Universal Robots PolyScope program: step2c_admittance_search30_z30_nostop_guard20_search2ms_line1ms_alpha70_v5.urp

Program step2c_admittance_search30_z30_nostop_guard20_search2ms_line1ms_alpha70_v5 (installation=default directory=/programs/andyl/kunwei/step2/step2c createdIn=5.11.9.1010452 lastSavedIn=5.11.9.1010452 robotSerialNumber=20225200364)
Calibrated DH parameters: a=[0.00002, -0.569483, -0.54992, -0.00001, -0.000036, 0]; d=[0.180894, -146.691669, 192.918669, -46.053088, 0.119778, 0.115602]; alpha=[1.571425, -0.001534, 0.003359, 1.568739, -1.571477, 0]; deltaTheta=[0, 0.376258, -0.101074, -0.275185, -0.000002, 0]
Robot Program (runOnlyOnce=true)
  Script file /programs/andyl/kunwei/step2/step2c/step2c/step2c_admittance_search30_z30_nostop_guard20_search2ms_line1ms_alpha70_v5.script
    | # Step2C admittance search30 v5: v4-style pre-contact approach with a 30-200 mm Z window, 50 percent lower normal admittance gain, and dynamic search-depth limit; TP-openable package.
    | # VERSION: 2026-06-08T1435HKT_STEP2C_V5_V4Z30_200_DAMP50_DEPTHFIX_NOFAILRETRACT
    | # GENERATED_AT_LOCAL: 2026-06-08T14:35:56+0800
    | # BEHAVIOR: wait for Kunwei bridge; align to old reference orientation; move to
    | # old contact-start XY; then bound the Z prep into old contact Z + 30..200 mm.
    | # If the current Z is already inside that window, keep it; otherwise move to the
    | # nearest bound and stop before search. Then search downward at 30 mm/s until 10 mm above known contact,
    | # 5 mm/s near the surface, using 2 ms speedl holds in both search and
    | # soft acquisition. Small-force early contact is gated to the near
    | # zone; far-zone unexpected contact requires larger raw force before entering
    | # soft acquisition targeting 2 N. The
    | # first 0.10 s of line control uses 10 ms speedl holds, then line control
    | # switches to 1 ms holds. Normal admittance P/I gains are reduced by 50 percent
    | # relative to the prior v4/v5 controller. Search-depth timeout is computed
    | # from the actual search-start Z so a 30-200 mm prep window can still search to
    | # 10 mm below known contact Z. A search-depth failure stops in place; it does
    | # not auto-retract upward.
    | # Aggressive normal Z correction targets signed Fz ~= -target_force_abs, where the bridge
    | # normally writes target_force_abs=5 N into input register 29.
    | # Raw contact triggers and safety guards remain unfiltered; only controller
    | # normal-velocity input uses a light force filter. No UR zero_ftsensor, no
    | # Kunwei tare/config write, no TCP/payload write, and no output register 34.
    | # Frequency contract: Kunwei raw may be about 1 kHz; RTDE handoff is requested
    | # at 500 Hz; search/admittance motion gate uses 2 ms speedl holds; line control
    | # switches to 1 ms holds after 0.10 s, but both phases must be measured before
    | # calling them 500 Hz authority. On successful completion only, retract 10 mm
    | # upward and then return to the TP-start home pose; failure paths do not auto-home.
    | 
    | def codex_abs(x):
    |   if x < 0.0:
    |     return -x
    |   end
    |   return x
    | end
    | 
    | def codex_clamp(x, lo, hi):
    |   if x < lo:
    |     return lo
    |   elif x > hi:
    |     return hi
    |   end
    |   return x
    | end
    | 
    | def codex_wait_for_sensor_ok(timeout_s):
    |   local dt = 0.002
    |   local t = 0.0
    |   while t < timeout_s:
    |     if read_input_float_register(27) > 0.5:
    |       return True
    |     end
    |     sync()
    |     t = t + dt
    |   end
    |   return False
    | end
    | 
    | def codex_wait_for_fresh_heartbeat(timeout_s):
    |   local dt = 0.002
    |   local t = 0.0
    |   local initial_heartbeat = read_input_float_register(26)
    |   local current_heartbeat = initial_heartbeat
    |   while t < timeout_s:
    |     current_heartbeat = read_input_float_register(26)
    |     write_output_float_register(26, current_heartbeat)
    |     write_output_float_register(35, 20.5)
    |     if read_input_float_register(27) > 0.5 and current_heartbeat != initial_heartbeat:
    |       return True
    |     end
    |     sync()
    |     t = t + dt
    |   end
    |   return False
    | end
    | 
    | def codex_step2_guard_stop_reason():
    |   local normal_force = read_input_float_register(24)
    |   local force_norm = read_input_float_register(25)
    |   local sensor_ok = read_input_float_register(27)
    |   local stop_request = read_input_float_register(28)
    |   local torque_norm = read_input_float_register(30)
    |   if sensor_ok < 0.5:
    |     return 3.0
    |   elif stop_request > 0.5:
    |     return 4.0
    |   elif codex_abs(normal_force) > 20.0:
    |     return 5.0
    |   elif force_norm > 50.0:
    |     return 6.0
    |   elif torque_norm > 0.6:
    |     return 7.0
    |   end
    |   return 0.0
    | end
    | 
    | def codex_write_echo(stop_reason, progress_m, correction_m, commanded_z_m_s):
    |   write_output_float_register(24, read_input_float_register(24))
    |   write_output_float_register(25, read_input_float_register(25))
    |   write_output_float_register(26, read_input_float_register(26))
    |   write_output_float_register(27, read_input_float_register(27))
    |   write_output_float_register(28, read_input_float_register(28))
    |   write_output_float_register(29, read_input_float_register(29))
    |   write_output_float_register(30, stop_reason)
    |   write_output_float_register(31, progress_m)
    |   write_output_float_register(32, correction_m)
    |   write_output_float_register(33, commanded_z_m_s)
    | end
    | 
    | def codex_step2c_full():
    |   local ux = 0.679764156
    |   local uy = -0.733430768
    |   local entry_x = 0.446585764
    |   local entry_y = 0.226717001
    |   local old_contact_z = 0.020279919
    |   local entry_z = old_contact_z + 0.100
    |   local ref_rx = 3.141572714
    |   local ref_ry = -0.000026465
    |   local ref_rz = -0.000024158
    |   local approach_speed_m_s = 0.080
    |   local approach_z_speed_m_s = 0.080
    |   local search_speed_m_s = -0.005
    |   local search_accel_m_s2 = 0.500
    |   local search_hold_s = 0.002
    |   local trigger_normal_force_n = -2.0
    |   local max_search_down_m = 0.110
    |   local stale_limit_s = 0.100
    |   local search_runtime_limit_s = 65.0
    |   local tangent_speed_m_s = 0.010
    |   local path_length_m = 0.06358
    |   local line_accel_m_s2 = 0.500
    |   local line_hold_s = 0.010
    |   local line_hold_fast_s = 0.001
    |   local line_fast_after_s = 0.100
    |   local line_runtime_limit_s = 15.0
    |   local target_force_abs_default_n = 5.0
    |   local normal_velocity_p_gain = 0.0003
    |   local normal_velocity_i_gain = 0.00004
    |   local normal_velocity_limit_m_s = 0.005
    |   local normal_filter_alpha = 0.70
    |   local integral_error_limit_n_s = 10.0
    |   local short_retract_z_m = 0.010
    |   local short_retract_speed_m_s = 0.020
    |   local home_return_speed_m_s = 0.080
    |   local stop_reason = 0.0
    |   local contact_triggered = 0
    |   local max_observed_stale_s = 0.0
    | 
    |   local home_pose = get_actual_tcp_pose()
    | 
    |   textmsg("codex step2c version 2026-06-08T1435HKT_STEP2C_V5_V4Z30_200_DAMP50_DEPTHFIX_NOFAILRETRACT start admittance_search30_v5_v4z30_200_damp50_depthfix_short_retract_home_return")
    |   write_output_float_register(35, 20.0)
    |   codex_write_echo(0.0, 0.0, 0.0, 0.0)
    | 
    |   if not codex_wait_for_fresh_heartbeat(30.0):
    |     stop_reason = 3.0
    |   end
    | 
    |   if stop_reason == 0.0:
    |     write_output_float_register(35, 21.0)
    |     local p0 = get_actual_tcp_pose()
    |     local reference_orientation_pose = p[p0[0], p0[1], p0[2], ref_rx, ref_ry, ref_rz]
    |     movel(reference_orientation_pose, a=0.030, v=approach_speed_m_s, r=0.0)
    |     stopl(0.5)
    |     write_output_float_register(35, 22.0)
    |     local p1 = get_actual_tcp_pose()
    |     local entry_xy_pose = p[entry_x, entry_y, p1[2], ref_rx, ref_ry, ref_rz]
    |     movel(entry_xy_pose, a=0.030, v=approach_speed_m_s, r=0.0)
    |     stopl(0.5)
    |     write_output_float_register(35, 23.0)
    |     local p2 = get_actual_tcp_pose()
    |     local max_entry_z = old_contact_z + 0.200
    |     local min_entry_z = old_contact_z + 0.030
    |     local bounded_entry_z = p2[2]
    |     if bounded_entry_z > max_entry_z:
    |       bounded_entry_z = max_entry_z
    |     elif bounded_entry_z < min_entry_z:
    |       bounded_entry_z = min_entry_z
    |     end
    |     if codex_abs(bounded_entry_z - p2[2]) > 0.002:
    |       local entry_pose = p[entry_x, entry_y, bounded_entry_z, ref_rx, ref_ry, ref_rz]
    |       movel(entry_pose, a=0.030, v=approach_z_speed_m_s, r=0.0)
    |       stopl(0.5)
    |     end
    |     sleep(0.20)
    |     stop_reason = codex_step2_guard_stop_reason()
    |   end
    | 
    |   if stop_reason == 0.0:
    |     write_output_float_register(35, 24.0)
    |     local search_start = get_actual_tcp_pose()
    |     max_search_down_m = search_start[2] - old_contact_z + 0.010
    |     if max_search_down_m < 0.040:
    |       max_search_down_m = 0.040
    |     elif max_search_down_m > 0.210:
    |       max_search_down_m = 0.210
    |     end
    |     local last_heartbeat = read_input_float_register(26)
    |     local stale_s = 0.0
    |     local t = 0.0
    |     local search_far_speed_m_s = -0.030
    |     local search_near_speed_m_s = -0.005
    |     local search_near_zone_m = 0.010
    |     local early_normal_force_n = -0.5
    |     local early_force_norm_n = 1.0
    |     local soft_target_force_n = 2.0
    |     local far_unexpected_normal_force_n = -5.0
    |     local far_unexpected_force_norm_n = 5.0
    |     local soft_acquire_p_gain = 0.0030
    |     local soft_velocity_limit_m_s = 0.008
    |     local soft_filter_alpha = 0.70
    |     local soft_enter_line_filtered_n = -1.8
    |     local soft_enter_line_raw_n = -2.0
    |     local soft_confirm_s = 0.030
    |     local early_contact = 0
    |     local stable_soft_s = 0.0
    |     local filtered_search_force = read_input_float_register(24)
    |     local commanded_search_z = search_far_speed_m_s
    |     while stop_reason == 0.0:
    |       local heartbeat = read_input_float_register(26)
    |       local normal_force = read_input_float_register(24)
    |       local force_norm = read_input_float_register(25)
    |       local pose_now = get_actual_tcp_pose()
    |       local search_depth_m = search_start[2] - pose_now[2]
    |       local height_above_known_contact_m = pose_now[2] - old_contact_z
    | 
    |       if heartbeat == last_heartbeat:
    |         stale_s = stale_s + search_hold_s
    |         if stale_s > max_observed_stale_s:
    |           max_observed_stale_s = stale_s
    |         end
    |       else:
    |         stale_s = 0.0
    |         last_heartbeat = heartbeat
    |       end
    | 
    |       if early_contact == 0:
    |         write_output_float_register(35, 24.0)
    |         if height_above_known_contact_m <= search_near_zone_m:
    |           if normal_force <= early_normal_force_n or force_norm > early_force_norm_n:
    |             early_contact = 1
    |             stable_soft_s = 0.0
    |             filtered_search_force = normal_force
    |             write_output_float_register(35, 24.4)
    |           end
    |         elif normal_force <= far_unexpected_normal_force_n or force_norm > far_unexpected_force_norm_n:
    |           early_contact = 1
    |           stable_soft_s = 0.0
    |           filtered_search_force = normal_force
    |           write_output_float_register(35, 24.4)
    |         end
    |       else:
    |         write_output_float_register(35, 24.4)
    |       end
    | 
    |       if stale_s > stale_limit_s:
    |         stop_reason = 2.0
    |       else:
    |         stop_reason = codex_step2_guard_stop_reason()
    |       end
    | 
    |       if stop_reason == 0.0:
    |         if search_depth_m >= max_search_down_m:
    |           stop_reason = 8.0
    |         elif t >= search_runtime_limit_s:
    |           stop_reason = 10.0
    |         else:
    |           if early_contact == 0:
    |             if height_above_known_contact_m > search_near_zone_m:
    |               commanded_search_z = search_far_speed_m_s
    |             else:
    |               commanded_search_z = search_near_speed_m_s
    |             end
    |             codex_write_echo(stop_reason, max_observed_stale_s, search_depth_m, commanded_search_z)
    |             speedl([0.0, 0.0, commanded_search_z, 0.0, 0.0, 0.0], search_accel_m_s2, search_hold_s)
    |             t = t + search_hold_s
    |           else:
    |             filtered_search_force = soft_filter_alpha * normal_force + (1.0 - soft_filter_alpha) * filtered_search_force
    |             local soft_force_error = soft_target_force_n + filtered_search_force
    |             commanded_search_z = 0.0 - codex_clamp(soft_acquire_p_gain * soft_force_error, -soft_velocity_limit_m_s, soft_velocity_limit_m_s)
    |             if filtered_search_force <= soft_enter_line_filtered_n or normal_force <= soft_enter_line_raw_n:
    |               stable_soft_s = stable_soft_s + search_hold_s
    |             else:
    |               stable_soft_s = 0.0
    |             end
    |             codex_write_echo(stop_reason, stable_soft_s, search_depth_m, commanded_search_z)
    |             if stable_soft_s >= soft_confirm_s:
    |               contact_triggered = 1
    |               stop_reason = 11.0
    |             else:
    |               speedl([0.0, 0.0, commanded_search_z, 0.0, 0.0, 0.0], search_accel_m_s2, search_hold_s)
    |               t = t + search_hold_s
    |             end
    |           end
    |         end
    |       end
    |     end
    |     stopl(0.5)
    | 
    |   end
    | 
    |   if contact_triggered == 1:
    |     stop_reason = 0.0
    |   end
    | 
    |   if stop_reason == 0.0:
    |     write_output_float_register(35, 25.0)
    |     local line_start = get_actual_tcp_pose()
    |     local last_heartbeat2 = read_input_float_register(26)
    |     local stale_s2 = 0.0
    |     local t2 = 0.0
    |     local filtered_normal_force = read_input_float_register(24)
    |     local integral_error = 0.0
    |     while stop_reason == 0.0:
    |       if t2 >= line_fast_after_s:
    |         line_hold_s = line_hold_fast_s
    |       end
    |       local raw_normal_force = read_input_float_register(24)
    |       local heartbeat2 = read_input_float_register(26)
    |       local target_force_abs = read_input_float_register(29)
    |       local pose_line = get_actual_tcp_pose()
    |       local dx = pose_line[0] - line_start[0]
    |       local dy = pose_line[1] - line_start[1]
    |       local progress_m = dx * ux + dy * uy
    |       local correction_m = pose_line[2] - line_start[2]
    | 
    |       if target_force_abs < 0.1:
    |         target_force_abs = target_force_abs_default_n
    |       end
    | 
    |       filtered_normal_force = normal_filter_alpha * raw_normal_force + (1.0 - normal_filter_alpha) * filtered_normal_force
    |       local force_error = target_force_abs + filtered_normal_force
    |       integral_error = codex_clamp(integral_error + force_error * line_hold_s, -integral_error_limit_n_s, integral_error_limit_n_s)
    |       local normal_velocity = 0.0 - codex_clamp(normal_velocity_p_gain * force_error + normal_velocity_i_gain * integral_error, -normal_velocity_limit_m_s, normal_velocity_limit_m_s)
    | 
    |       if heartbeat2 == last_heartbeat2:
    |         stale_s2 = stale_s2 + line_hold_s
    |       else:
    |         stale_s2 = 0.0
    |         last_heartbeat2 = heartbeat2
    |       end
    | 
    |       codex_write_echo(stop_reason, progress_m, correction_m, normal_velocity)
    | 
    |       if stale_s2 > stale_limit_s:
    |         stop_reason = 2.0
    |       else:
    |         stop_reason = codex_step2_guard_stop_reason()
    |       end
    | 
    |       if stop_reason == 0.0:
    |         if codex_abs(correction_m) > 0.008:
    |           stop_reason = 8.0
    |         elif progress_m < -0.003 or progress_m > 0.067:
    |           stop_reason = 9.0
    |         elif t2 >= line_runtime_limit_s:
    |           stop_reason = 10.0
    |         elif progress_m >= path_length_m:
    |           stop_reason = 1.0
    |         else:
    |           speedl([ux * tangent_speed_m_s, uy * tangent_speed_m_s, normal_velocity, 0.0, 0.0, 0.0], line_accel_m_s2, line_hold_s)
    |           t2 = t2 + line_hold_s
    |         end
    |       end
    |     end
    |     stopl(0.5)
    |   end
    | 
    |   if stop_reason == 1.0:
    |     write_output_float_register(35, 26.0)
    |     local short_retract_start = get_actual_tcp_pose()
    |     local short_retract_pose = p[short_retract_start[0], short_retract_start[1], short_retract_start[2] + short_retract_z_m, short_retract_start[3], short_retract_start[4], short_retract_start[5]]
    |     codex_write_echo(stop_reason, path_length_m, short_retract_z_m, 0.0)
    |     movel(short_retract_pose, a=0.030, v=short_retract_speed_m_s, r=0.0)
    |     stopl(0.5)
    |     write_output_float_register(35, 27.0)
    |     codex_write_echo(stop_reason, path_length_m, short_retract_z_m, 0.0)
    |     movel(home_pose, a=0.030, v=home_return_speed_m_s, r=0.0)
    |     stopl(0.5)
    |   end
    | 
    |   write_output_float_register(30, stop_reason)
    |   write_output_float_register(31, max_observed_stale_s)
    |   write_output_float_register(35, 29.0)
    |   textmsg("codex step2c version 2026-06-08T1435HKT_STEP2C_V5_V4Z30_200_DAMP50_DEPTHFIX_NOFAILRETRACT stop reason:", stop_reason)
    | end
    | 
    | codex_step2c_full()
